Staubli VAL3: Vakuumgreifer.pjx

--- Vakuumgreifer.pjx ---
Parameters version=s7.5.3 stackSize=5000 millimeterUnit=true
Program file=MoveJoint.pgx
Program file=MoveLine.pgx
Program file=start.pgx
Program file=stop.pgx
Program file=main.pgx
Data file=Vakuumgreifer.dtx

--- Vakuumgreifer.dtx ---
frame StaubliTX240Base = {x=0.000, y=0.000, z=0.000, rx=-0.000, ry=0.000, rz=-0.000, fatherId=world[0]}
dio dVacuum = {link=98FE10BA-0446-4B8A-A8CF-35B98F42725A}
tool tCurrentTool = {x=0.000, y=0.000, z=78.000, rx=-0.000, ry=0.000, rz=-0.000, fatherId=flange[0], ioLink=98FE10BA-0446-4B8A-A8CF-35B98F42725A}
mdesc mCurrentSpeed
pointRx pPointRx1 = {}
pointRx pPointRx2 = {}

--- main.pgx ---
program main()
begin
		close(tCurrentTool)
    pPointRx1.config.shoulder = lefty
    pPointRx1.config.elbow = epositive
    pPointRx1.config.wrist = wpositive
    pPointRx2.config.shoulder = lefty
    pPointRx2.config.elbow = epositive
    pPointRx2.config.wrist = wpositive
    mCurrentSpeed.tvel = 100.00
    mCurrentSpeed.blend = joint
    mCurrentSpeed.reach = 0.010
    mCurrentSpeed.leave = 0.010
    		// Program Vakuumgreifer start
		// Program generated by RoboDK v5.2.1 for Staubli TX2-40 on 26/04/2021 14:08:58
		link(pPointRx1,StaubliTX240Base)
		link(pPointRx2,StaubliTX240Base)
		call MoveJoint(0.00000,45.00000,45.00000,0.00000,90.00000,0.00000)
		call MoveJoint(-14.60130,45.44290,110.13300,0.00000,24.42430,-14.60130)
		call MoveJoint(-28.98340,73.16320,77.29560,0.00000,29.54110,-28.54940)
		call MoveLine(302.386,-127.490,-323.580,-180.000,0.000,-179.566)
		waitEndMove()
		dioSet(dVacuum[0],1.000000)
		call MoveLine(302.386,-127.490,-273.580,-180.000,0.000,-179.566)
		call MoveJoint(-14.60130,45.44290,110.13300,0.00000,24.42430,-14.60130)
		call MoveJoint(-28.98340,73.16320,77.29560,0.00000,29.54110,-28.54940)
		call MoveLine(302.386,-127.490,-323.580,-180.000,0.000,-179.566)
		waitEndMove()
		dioSet(dVacuum[0],0.000000)
		call MoveJoint(0.00000,45.00000,45.00000,0.00000,90.00000,0.00000)

		waitEndMove()
		// Program Vakuumgreifer end

end

--- MoveLine.pgx ---
program MoveLine(num x_nX, num x_nY, num x_nZ, num x_nRx, num x_nRy, num x_nRz)
begin
  pPointRx1.trsf.x = x_nX
  pPointRx1.trsf.y = x_nY
  pPointRx1.trsf.z = x_nZ
  pPointRx1.trsf.rx = x_nRx
  pPointRx1.trsf.ry = x_nRy
  pPointRx1.trsf.rz = x_nRz
  movel(pPointRx1,tCurrentTool,mCurrentSpeed)
end
